// TIA Portal V20 export
VAR_GLOBAL   // PLC tag table "AddOn"
END_VAR
VAR_GLOBAL CONSTANT   // user constants
   STS_ABORTING : DInt := 1;   // Machine state Aborting
   STS_ABORTED : DInt := 2;   // Machine state Aborted
   STS_STOPPING : DInt := 3;   // Machine state Stopping
   STS_STOPPED : DInt := 4;   // Machine state Stopped
   STS_RESETTING : DInt := 5;   // Machine state Resetting
   STS_IDLE : DInt := 6;   // Machine state Idle
   STS_STARTING : DInt := 7;   // Machine state Starting
   STS_EXECUTE : DInt := 8;   // Machine state Execute
   STS_HOLDING : DInt := 9;   // Machine state Holding
   STS_HELD : DInt := 10;   // Machine state Held
   STS_SUSPENDING : DInt := 11;   // Machine state Suspending
   STS_SUSPENDED : DInt := 12;   // Machine state Suspended
   LACYCCOM_WRITE_PARAMETERS_UPPER_LIM : Int := 18;   // Upper limit of write parameters
   LACYCCOM_READ_PARAMETERS_UPPER_LIM : Int := 38;   // Upper limit of read parameters
   LACYCCOM_SILENT_OPERATION_PARAMETERS_UPPER_LIM : Int := 17;   // Upper limit of parameters in LAcycCom_typeDriveSilentOperation
   LACYCCOM_NO_COMMAND : Byte := 16#00;   // No command
   LACYCCOM_READ_COMMAND : Byte := 16#01;   // Read command
   LACYCCOM_WRITE_COMMAND : Byte := 16#02;   // Write command
   LACYCCOM_TYPE_ALARM : SInt := 1;   // Alarm
   LACYCCOM_TYPE_FAULT : SInt := 2;   // Fault
   LACYCCOM_TYPE_SI_MESSAGE : SInt := 3;   // SI message
   LACYCCOM_MESSAGES_UPPER_LIM : Int := 23;   // Upper limit of elements in LAcycCom_typeDriveMessages (fix value)
   LACYCCOM_BUFFER_ELEMENTS_UPPER_LIM : Int := 59;   // Upper limit of buffer elements
   Cfg_XTS_NbrMaxPosition : DInt := 256;   // Maximum number of Positions
   Cfg_XTS_NbrMaxMover : DInt := 200;   // Maximum number of Movers
   Cfg_XTS_NbrOfHMI_Interface : DInt := 10;   // Number of HMI Interfaces
   Cfg_XTS_MaxSyncLoop : DInt := 40;   // Maximum number of Positions for one station
END_VAR
